// TIA Portal V20 export
DATA_BLOCK "LBP_Internal2"   // DB25001
TITLE = Internal DB for basic program / DB interne pour programme de base
// DB only for internal use in the basic program / DB réservé à l'utilisation interne dans le programme de base
// stored: InstanceOfName LBP_InternalProc7, InstanceOfType FB
"LBP_InternalProc7"
   // VAR_OUTPUT
   //    error { ExternalAccessible := 'False'; ExternalVisible := 'False'; ExternalWritable := 'False'} : Bool;
   // END_VAR
   // VAR
   //    statTimer1 { ExternalAccessible := 'False'; ExternalVisible := 'False'; ExternalWritable := 'False'} : Array[1..8] of IEC_TIMER;
   //    statTimer2 { ExternalAccessible := 'False'; ExternalVisible := 'False'; ExternalWritable := 'False'} : Array[1..8] of IEC_TIMER;
   //    statTimerActivationImmediately { ExternalAccessible := 'False'; ExternalVisible := 'False'; ExternalWritable := 'False'} : Array[1..8] of IEC_TIMER;   // Delay time for immediate activation / Temporisation pour activation immédiate
   //    statActivationImmediately { ExternalAccessible := 'False'; ExternalVisible := 'False'; ExternalWritable := 'False'} : Array[1..8] of Bool;
   //    statImpReloadT2 { ExternalAccessible := 'False'; ExternalVisible := 'False'; ExternalWritable := 'False'} : Array[1..8] of R_TRIG;
   //    statMcp1 { ExternalAccessible := 'False'; ExternalVisible := 'False'; ExternalWritable := 'False'} : Array[0..1, 0..7] of Byte;   // Image of mcp1 to detect any changes / Image de la mcp1 pour comparaison
   //    statMcp2 { ExternalAccessible := 'False'; ExternalVisible := 'False'; ExternalWritable := 'False'} : Array[0..1, 0..7] of Byte;   // Image of mcp2 to detect any changes / Image de la mcp2 pour comparaison
   //    statTimerDataTranfer { ExternalAccessible := 'False'; ExternalVisible := 'False'; ExternalWritable := 'False'} : IEC_TIMER;
   //    statChanInReset { ExternalAccessible := 'False'; ExternalVisible := 'False'; ExternalWritable := 'False'} : Array[1..10] of Bool;
   //    statAktProfile { ExternalAccessible := 'False'; ExternalVisible := 'False'; ExternalWritable := 'False'} : Struct
   //       ESaveOn : Bool;   // Activate energy-saving profile immediately / Activer immédiatement le profil d'économie d'énergie
   //       ReloadT2 : Bool;   // Reload Prewarning time (T2) / Recharger temps de préavis (T2)
   //       res0_2 : Bool;
   //       res0_3 : Bool;
   //       res0_4 : Bool;
   //       res0_5 : Bool;
   //       res0_6 : Bool;
   //       res0_7 : Bool;
   //       HmiESaveOn : Bool;   // HMI->PLC: Activate energy-saving profile immediately / IHM->AP : activer immédiatement le profil d'économie d'énergie
   //       res1_1 : Bool;
   //       res1_2 : Bool;
   //       res1_3 : Bool;
   //       res1_4 : Bool;
   //       res1_5 : Bool;
   //       res1_6 : Bool;
   //       res1_7 : Bool;
   //       MasterCompSig : Bool;   // Master computer signal / Signal ordinateur maître
   //       PlcUserSig : Bool;   // PLC user signal / AP signal utilisateur
   //       res2_2 : Bool;
   //       res2_3 : Bool;
   //       res2_4 : Bool;
   //       res2_5 : Bool;
   //       res2_6 : Bool;
   //       res2_7 : Bool;
   //       res3 : Byte;
   //       ESaveIsOn : Bool;   // Energy-saving state active / État économie d'énergie actif
   //       T1Expired : Bool;   // Activation time T1 expired / Temps d'activation T1 écoulé
   //       res4_2 : Bool;
   //       res4_3 : Bool;
   //       res4_4 : Bool;
   //       res4_5 : Bool;
   //       res4_6 : Bool;
   //       res4_7 : Bool;
   //       res5 : Byte;
   //       ActValT1 : Int;   // T1 current value / T1 valeur réelle
   //       ActValT2 : Int;   // T2 current value / T2 valeur réelle
   //       ESaveValid : Bool;   // HMI->PLC: Energy-saving profile valid / IHM->AP : profil d'économie d'énergie valide
   //       ESaveOff : Bool;   // HMI->PLC: Deactivate energy-saving profileblock energy-saving profile / IHM->AP : désactiver/bloquer le profil d'économie d'énergie
   //       res10_2 : Bool;
   //       res10_3 : Bool;
   //       res10_4 : Bool;
   //       res10_5 : Bool;
   //       res10_6 : Bool;
   //       res10_7 : Bool;
   //       CondOpPanel : Bool;   // HMI->PLC: Operator panel / IHM->AP : pupitre opérateur
   //       CondDataTransfer : Bool;   // HMI->PLC: Data transfer / IHM->AP : transmission de données
   //       CondWindowChange : Bool;   // HMI->PLC: Window change / IHM->AP : changement de fenêtre
   //       res11_3 : Bool;
   //       res11_4 : Bool;
   //       res11_5 : Bool;
   //       res11_6 : Bool;
   //       res11_7 : Bool;
   //       CondMCP : Bool;   // HMI->PLC: Machine control panel / IHM->AP : pupitre opérateur machine
   //       res12_1 : Bool;
   //       res12_2 : Bool;
   //       res12_3 : Bool;
   //       res12_4 : Bool;
   //       res12_5 : Bool;
   //       res12_6 : Bool;
   //       res12_7 : Bool;
   //       CondNcChan1 : Bool;   // HMI->PLC: NC channel 1 in reset / IHM->AP : canal CN 1 en Reset
   //       CondNcChan2 : Bool;   // HMI->PLC: NC channel 2 in reset / IHM->AP : canal CN 2 en Reset
   //       CondNcChan3 : Bool;   // HMI->PLC: NC channel 3 in reset / IHM->AP : canal CN 3 en Reset
   //       CondNcChan4 : Bool;   // HMI->PLC: NC channel 4 in reset / IHM->AP : canal CN 4 en Reset
   //       CondNcChan5 : Bool;   // HMI->PLC: NC channel 5 in reset / IHM->AP : canal CN 5 en Reset
   //       CondNcChan6 : Bool;   // HMI->PLC: NC channel 6 in reset / IHM->AP : canal CN 6 en Reset
   //       CondNcChan7 : Bool;   // HMI->PLC: NC channel 7 in reset / IHM->AP : canal CN 7 en Reset
   //       CondNcChan8 : Bool;   // HMI->PLC: NC channel 8 in reset / IHM->AP : canal CN 8 en Reset
   //       CondNcChan9 : Bool;   // HMI->PLC: NC channel 9 in reset / IHM->AP : canal CN 9 en Reset
   //       CondNcChan10 : Bool;   // HMI->PLC: NC channel 10 in reset / IHM->AP : canal CN 10 en Reset
   //       res14_2 : Bool;
   //       res14_3 : Bool;
   //       res14_4 : Bool;
   //       res14_5 : Bool;
   //       res14_6 : Bool;
   //       res14_7 : Bool;
   //       CondMasterCompSig : Bool;   // HMI->PLC: Master computer signal / IHM->AP : signal ordinateur maître
   //       CondPlcUserSig : Bool;   // HMI->PLC: PLC user signal / IHM->AP : signal utilisateur AP
   //       res15_2 : Bool;
   //       res15_3 : Bool;
   //       res15_4 : Bool;
   //       res15_5 : Bool;
   //       res15_6 : Bool;
   //       res15_7 : Bool;
   //       PresetT1 : Int;   // HMI->PLC: Activation time T1 / IHM->AP : temps d'activation T1
   //       PresetT2 : Int;   // HMI->PLC: Activation time T2 / IHM->AP : temps d'activation T2
   //    END_STRUCT;
   // END_VAR
BEGIN
END_DATA_BLOCK
